SUBAPPLICATION INI_IN_AND_STORE_UDINT (* DigitalInput_I1 auf DigitalOutput_Q1; E_TON Einschaltverzögert; Zeit eingeben und speichern, INI *)
  (* Standard: 61499-2; Description: Copyright (c) 2023 Meisterschulen am Ostbahnhof This program and the accompanying materials are made available under the terms of the Eclipse Public License 2.0 which is available at https://www.eclipse.org/legal/epl-2.0/ SPDX-License-Identifier: EPL-2.0 *)
  (* Version 1.0, 2023-10-31, Franz Höpfinger, Meisterschulen am Ostbahnhof, initial API and implementation and/or initial documentation *)
  PACKAGE MyLib::sys;
  IMPORT isobus::UT::Q::const::IDs::ID_NULL;
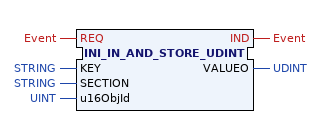
  EVENT_INPUT
    REQ;
  END_EVENT
  EVENT_OUTPUT
    IND;
  END_EVENT
  VAR_INPUT
    KEY : STRING; (* Key name. *)
    SECTION : STRING; (* Section name. *)
    u16ObjId : UINT := ID_NULL;
  END_VAR
  VAR_OUTPUT
    VALUEO : UDINT;
  END_VAR
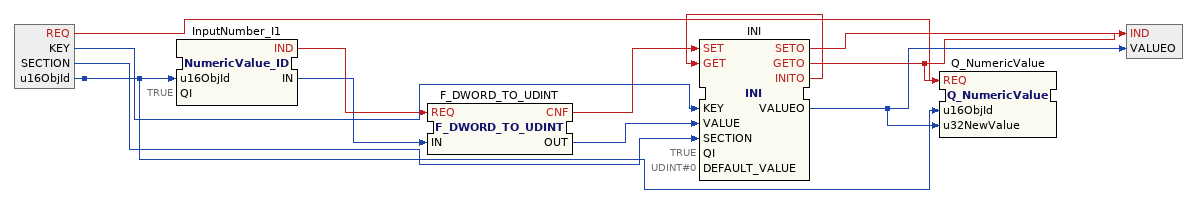
  FBS
    InputNumber_I1 : isobus::UT::io::NumericValue::NumericValue_ID(QI := TRUE);
    F_DWORD_TO_UDINT : iec61131::conversion::F_DWORD_TO_UDINT;
    INI : eclipse4diac::storage::INI(QI := TRUE, DEFAULT_VALUE := UDINT#0);
    Q_NumericValue : isobus::UT::Q::Q_NumericValue;
  END_FBS
  EVENT_CONNECTIONS
    InputNumber_I1.IND TO F_DWORD_TO_UDINT.REQ;
    REQ TO Q_NumericValue.REQ;
    F_DWORD_TO_UDINT.CNF TO INI.SET;
    INI.SETO TO IND;
    INI.GETO TO Q_NumericValue.REQ;
    INI.GETO TO IND;
    INI.INITO TO INI.GET;
  END_CONNECTIONS
  DATA_CONNECTIONS
    InputNumber_I1.IN TO F_DWORD_TO_UDINT.IN;
    u16ObjId TO Q_NumericValue.u16ObjId;
    KEY TO INI.KEY;
    F_DWORD_TO_UDINT.OUT TO INI.VALUE;
    INI.VALUEO TO Q_NumericValue.u32NewValue;
    INI.VALUEO TO VALUEO;
    u16ObjId TO InputNumber_I1.u16ObjId;
    SECTION TO INI.SECTION;
  END_CONNECTIONS
END_SUBAPPLICATION
